FUNCTION_BLOCK STYLE_AND (* Composite Function Block Type *)
  (* Standard: 61499-2 *)
  (* Version 0.2, 2003-12-05, JHC, Rockwell Automation, Renamed from NEWCOMPFB. *)
  (* Version 0.1, 2002-01-08, JHC, Rockwell Automation, Added DLY FB as example. *)
  (* Version 0.0, 2000-05-27, JHC, Rockwell Automation *)
  (* Compiler header: package fb.rt.student; *)
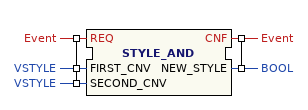
  EVENT_INPUT
    REQ WITH FIRST_CNV, SECOND_CNV; (* Normal Execution Request *)
  END_EVENT
  EVENT_OUTPUT
    CNF WITH NEW_STYLE; (* Execution Confirmation *)
  END_EVENT
  VAR_INPUT
    FIRST_CNV : VSTYLE;
    SECOND_CNV : VSTYLE;
  END_VAR
  VAR_OUTPUT
    NEW_STYLE : BOOL;
  END_VAR
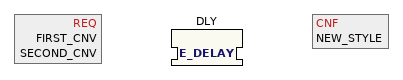
  FBS
    DLY : E_DELAY;
  END_FBS
END_FUNCTION_BLOCK
